(* IEC 61131-3 sources: volt/packages/volt-lsp-iec/test-corpus/pro2193/Device/Plc Logic/Application/04 Physical Interfaces/Ethernet/13 Dashboard/EdgePcClient, 2 files *)

(* ---- ProductionStatisticListenerFB.pou ---- *)
{attribute 'call_after_init'}
FUNCTION_BLOCK PUBLIC ProductionStatisticListenerFB
IMPLEMENTS IObserver
VAR_INPUT
	subject						: ISubject;
	edgePcClient				: IAddLog;
END_VAR
VAR
	ProductionCountersConfig	: EdgePcLogging.ProductionCountersPlcDataTypesConfig;
END_VAR

%LANGUAGE ST
Initialize();

END_FUNCTION_BLOCK

METHOD PRIVATE Initialize
VAR_INST
	{attribute 'init_on_onlchange' }
	initialized	: BOOL;
END_VAR

%LANGUAGE ST
IF initialized THEN
	RETURN;
END_IF

subject.Attach(THIS^);

EdgePcLogging.GenerateProductionCountersPlcDataTypesConfig(countersConfig := ProductionCountersConfig);

initialized := TRUE;

END_METHOD

// The Update method is called when subjects have a new state
METHOD Update
VAR_INPUT
	payload			: ISubjectBasePayload;
END_VAR
VAR
	stat			: ISubjectProductionStatistic;
	plcDataType1	: PlcDataType;
END_VAR

%LANGUAGE ST
// Check if we receive the right kind of data
IF NOT __QUERYINTERFACE(payload, stat) THEN
	RETURN;
END_IF

//Disable warning C0327: Implicit conversion from one enumeration type (PLCDATATYPE) to another (PLCDATATYPE (edgepclogging, x.x (brink automation)))
{warning disable C0327}

CASE stat.StatType OF
	enumProductionStatsCavityType.Produced:				plcDataType1 := productionCountersConfig[stat.Cavity].Produced;
	enumProductionStatsCavityType.Stacked:				plcDataType1 := productionCountersConfig[stat.Cavity].Stacked;
	enumProductionStatsCavityType.Rejected:				plcDataType1 := productionCountersConfig[stat.Cavity].Rejected;
	enumProductionStatsCavityType.UncountedReject:		plcDataType1 := productionCountersConfig[stat.Cavity].UncountedReject;
	enumProductionStatsCavityType.RejectReason:			plcDataType1 := productionCountersConfig[stat.Cavity].RejectReasons[stat.RejectReason - 1]; // Lelijk, in library oplossen!!
END_CASE

edgePcClient.AddLogLINT(	plcDataType	:= plcDataType1,
							value		:= stat.Data);

{warning restore C0327}

END_METHOD

(* ---- EdgePcPrg.pou ---- *)
PROGRAM EdgePcPrg
VAR
	client							: EdgePcLogging.EdgePcClient;
	taskInterval					: BYTE;
	logCache						: EdgePcLogging.LogCache;		// INTERNAL use only! Please use 'client' to log data!
	stringLogCache					: EdgePcLogging.StringLogCache;	// INTERNAL use only! Please use 'client' to log data!
	ConnectDelay					: BTON;
	connectToEdgePcClient			: BOOL := TRUE;
	{attribute 'init_on_onlchange' }
	forceReconnectOnOnlineChange	: BOOL := TRUE;

	ProductionStatisticListener		: ProductionStatisticListenerFB;

	taskInfo				: CmpIecTask.Task_Info2;

END_VAR

%LANGUAGE ST
__TRY
taskInfo	:= TaskGetInfo();

IF NOT Initialize() THEN
	RETURN;
END_IF

client(
	connect			:= ConnectDelay.Set(connectToEdgePcClient AND NOT forceReconnectOnOnlineChange, 2),
	ipv4Address		:= HMI.ipAddressEdgePC,
	port			:= HMI.communicationPortEdgePC,
	serSerialNo		:= HMI.robotSerial,
	logCache		:= logCache,
	stringLogCache	:= stringLogCache,
	connSpeed		:= ConnectionSpeed.S100Mbps,
	cycleMs			:= taskInterval // Verify that this value is the cycle interval of the EdgePcTask!
);

forceReconnectOnOnlineChange R= forceReconnectOnOnlineChange;

ProductionStatisticListener(
		subject			:= SER.Statistics,
		edgePcClient	:= client,
);

__CATCH(GVL_Exceptions.aeExceptionCodes[eExceptionCodes.EdgePcTask])
	GVL_Exceptions.xException := TRUE;
	GVL_Exceptions.iCounter := GVL_Exceptions.iCounter + 1;
__ENDTRY

END_PROGRAM

METHOD PRIVATE Initialize : BOOL
VAR_INST
	{attribute 'init_on_onlchange'}
	initialized	: BOOL;
END_VAR

%LANGUAGE ST
IF initialized THEN
	Initialize		:= TRUE;
	RETURN;
END_IF

taskInterval		:= TO_BYTE(TaskGetInterval());

IF NOT Stu.StrIsNullOrEmptyA(ADR(HMI.robotSerial))
AND taskInterval <> 0
THEN
	initialized		:= TRUE;
	Initialize		:= TRUE;
END_IF

END_METHOD
